// TIA Portal project "CIP" (V17)

(* hardware
DEVICE "S7-1200 station_1"  S7-1200 Station
   slot 0: "Rack_0"  S7-1200 Rack  Rack  V1.0
   slot 1: "PLC_1"  CPU 1214C DC/DC/DC  6ES7 214-1AG40-0XB0  V4.5
   slot 2: "AI 4x13BIT/AQ 2x14BIT_1"  6ES7 234-4HE32-0XB0  V2.1
   slot 3: "DI 16/DQ 16x24VDC_1"  6ES7 223-1BL32-0XB0  V2.0
DEVICE "HMI_1"  KTP600 Basic mono PN
   slot 0: "HMI_1"  KTP600 Basic mono PN  6AV6 647-0AB11-3AX0  12.0.0.0
   slot 1: "HMI_RT_1"  KTP600 Basic mono PN  6AV6 647-0AB11-3AX0  12.0.0.0
   slot 5: "HMI_1.IE_CP_1"  PROFINET Interface  12.0.0.0
      slot 1: "PROFINET Interface_1"  PROFINET Interface
         slot 1: "Port_1"  Port
*)

// ===== PLC "PLC_1"  CPU 1214C DC/DC/DC =====

VAR_GLOBAL   // PLC tag table "Default tag table"
   "VALVE_WASHABLE_DEVICE_INPUT" AT %Q1000.0 : Bool;
   "VALVE_WASHABLE_DEVICE_BACK" AT %Q1000.1 : Bool;
   "VALVE_INTERMEDIATE_1" AT %Q1000.2 : Bool;
   "VALVE_WATER_INPUT" AT %Q1000.3 : Bool;
   "VALVE_WATER_OUTPUT" AT %Q1000.4 : Bool;
   "VALVE_INTERMEDIATE_2" AT %Q1001.0 : Bool;
   "VALVE_INTERMEDIATE_3" AT %Q1001.1 : Bool;
   "VALVE_INTERMEDIATE_4" AT %Q1001.2 : Bool;
   "VALVE_WATER_TANK_INPUT" AT %Q1001.3 : Bool;
   "VALVE_WATER_TANK_INPUT_CLEAN" AT %Q1001.4 : Bool;
   "VALVE_WATER_TANK_OUTPUT" AT %Q1001.5 : Bool;
   "VALVE_ALKALI_TANK_INPUT" AT %Q1001.6 : Bool;
   "VALVE_ALKALI_TANK_INPUT_CLEAN" AT %Q1001.7 : Bool;
   "VALVE_ALKALI_TANK_OUTPUT" AT %Q1002.0 : Bool;
   "VALVE_ACID_TANK_INPUT" AT %Q1002.1 : Bool;
   "VALVE_ACID_TANK_INPUT_CLEAN" AT %Q1002.2 : Bool;
   "VALVE_ACID_TANK_OUTPUT" AT %Q1002.3 : Bool;
   "VALVE_STEAM" AT %Q1002.4 : Bool;
   "PUMP" AT %Q1002.5 : Bool;
   "BACK_PUMP" AT %Q1002.6 : Bool;
END_VAR

DATA_BLOCK "MAIN_DB"   // DB1
{ S7_Optimized_Access := 'TRUE' }
VERSION : 0.1
// stored: InstanceOfName MAIN
"MAIN"
BEGIN
END_DATA_BLOCK

DATA_BLOCK "ACTUATORS_DB"   // DB2
{ S7_Optimized_Access := 'TRUE' }
VERSION : 0.1
// stored: InstanceOfName ACTUATORS
"ACTUATORS"
BEGIN
END_DATA_BLOCK

DATA_BLOCK "VALVES_AND_PUMPS_STATES_DB"   // DB3
{ S7_Optimized_Access := 'TRUE' }
VERSION : 0.1
// stored: InstanceOfName VALVES_AND_PUMPS_STATES
"VALVES_AND_PUMPS_STATES"
BEGIN
END_DATA_BLOCK

FUNCTION_BLOCK "MAIN"   // FB1, SCL
{ S7_Optimized_Access := 'TRUE' }
VERSION : 0.1
BEGIN

   "VALVES_AND_PUMPS_STATES_DB"();

   "ACTUATORS_DB"();
END_FUNCTION_BLOCK

FUNCTION_BLOCK "ACTUATORS"   // FB2, SCL
{ S7_Optimized_Access := 'TRUE' }
VERSION : 0.1
   VAR
      VALVE_WASHABLE_DEVICE_INPUT : "ACTUATOR";
      VALVE_WASHABLE_DEVICE_BACK : "ACTUATOR";
      VALVE_INTERMEDIATE_1 : "ACTUATOR";
      VALVE_WATER_INPUT : "ACTUATOR";
      VALVE_WATER_OUTPUT : "ACTUATOR";
      VALVE_INTERMEDIATE_2 : "ACTUATOR";
      VALVE_INTERMEDIATE_3 : "ACTUATOR";
      VALVE_INTERMEDIATE_4 : "ACTUATOR";
      VALVE_WATER_TANK_INPUT : "ACTUATOR";
      VALVE_WATER_TANK_INPUT_CLEAN : "ACTUATOR";
      VALVE_WATER_TANK_OUTPUT : "ACTUATOR";
      VALVE_ALKALI_TANK_INPUT : "ACTUATOR";
      VALVE_ALKALI_TANK_INPUT_CLEAN : "ACTUATOR";
      VALVE_ALKALI_TANK_OUTPUT : "ACTUATOR";
      VALVE_ACID_TANK_INPUT : "ACTUATOR";
      VALVE_ACID_TANK_INPUT_CLEAN : "ACTUATOR";
      VALVE_ACID_TANK_OUTPUT : "ACTUATOR";
      VALVE_STEAM : "VALVE_STEAM1";
      PUMP : "ACTUATOR";
      BACK_PUMP : "ACTUATOR";
   END_VAR
BEGIN

   #VALVE_WASHABLE_DEVICE_INPUT("VALVE_WASHABLE_DEVICE_INPUT");

   #VALVE_WASHABLE_DEVICE_BACK("VALVE_WASHABLE_DEVICE_BACK");

   #VALVE_INTERMEDIATE_1("VALVE_INTERMEDIATE_1");

   #VALVE_WATER_INPUT("VALVE_WATER_INPUT");

   #VALVE_WATER_OUTPUT("VALVE_WATER_OUTPUT");

   #VALVE_INTERMEDIATE_2("VALVE_INTERMEDIATE_2");

   #VALVE_INTERMEDIATE_3("VALVE_INTERMEDIATE_3");

   #VALVE_INTERMEDIATE_4("VALVE_INTERMEDIATE_4");

   #VALVE_WATER_TANK_INPUT("VALVE_WATER_TANK_INPUT");

   #VALVE_WATER_TANK_INPUT_CLEAN("VALVE_WATER_TANK_INPUT_CLEAN");

   #VALVE_WATER_TANK_OUTPUT("VALVE_WATER_TANK_OUTPUT");

   #VALVE_ALKALI_TANK_INPUT("VALVE_ALKALI_TANK_INPUT");

   #VALVE_ALKALI_TANK_INPUT_CLEAN("VALVE_ALKALI_TANK_INPUT_CLEAN");

   #VALVE_ALKALI_TANK_OUTPUT("VALVE_ALKALI_TANK_OUTPUT");

   #VALVE_ACID_TANK_INPUT("VALVE_ACID_TANK_INPUT");

   #VALVE_ACID_TANK_INPUT_CLEAN("VALVE_ACID_TANK_INPUT_CLEAN");

   #VALVE_ACID_TANK_OUTPUT("VALVE_ACID_TANK_OUTPUT");

   #VALVE_STEAM();

   #PUMP("PUMP");

   #BACK_PUMP("BACK_PUMP");
END_FUNCTION_BLOCK

FUNCTION_BLOCK "ACTUATOR"   // FB3, SCL
{ S7_Optimized_Access := 'TRUE' }
VERSION : 0.1
   VAR_OUTPUT
      OUTPUT : Bool;
   END_VAR
   VAR
      MODE : Int;
      AUTO_VALUE : Bool;
   END_VAR
BEGIN
   CASE #MODE OF
       0:
           #OUTPUT := FALSE;
       1:
           #OUTPUT := TRUE;
       2:
           #OUTPUT := #AUTO_VALUE;
   END_CASE;
END_FUNCTION_BLOCK

FUNCTION_BLOCK "VALVES_AND_PUMPS_STATES"   // FB4, SCL
{ S7_Optimized_Access := 'TRUE' }
VERSION : 0.1
   VAR
      STATE : Int;
      VALVE_WASHABLE_DEVICE_BACK_STATES : Array[0..26] of Bool;
      VALVE_WASHABLE_DEVICE_INPUT_STATES : Array[0..26] of Bool;
      VALVE_INTERMEDIATE_1_STATES : Array[0..26] of Bool;
      VALVE_WATER_INPUT_STATES : Array[0..26] of Bool;
      VALVE_WATER_OUTPUT_STATES : Array[0..26] of Bool;
      VALVE_INTERMEDIATE_2_STATES : Array[0..26] of Bool;
      VALVE_INTERMEDIATE_3_STATES : Array[0..26] of Bool;
      VALVE_INTERMEDIATE_4_STATES : Array[0..26] of Bool;
      VALVE_WATER_TANK_INPUT_STATES : Array[0..26] of Bool;
      VALVE_WATER_TANK_INPUT_CLEAN_STATES : Array[0..26] of Bool;
      VALVE_WATER_TANK_OUTPUT_STATES : Array[0..26] of Bool;
      VALVE_ALKALI_TANK_INPUT_STATES : Array[0..26] of Bool;
      VALVE_ALKALI_TANK_INPUT_CLEAN_STATES : Array[0..26] of Bool;
      VALVE_ALKALI_TANK_OUTPUT_STATES : Array[0..26] of Bool;
      VALVE_ACID_TANK_INPUT_STATES : Array[0..26] of Bool;
      VALVE_ACID_TANK_INPUT_CLEAN_STATES : Array[0..26] of Bool;
      VALVE_ACID_TANK_OUTPUT_STATES : Array[0..26] of Bool;
      PUMP_STATES : Array[0..26] of Bool;
      BACK_PUMP_STATES : Array[0..26] of Bool;
   END_VAR
   // VALVE_WASHABLE_DEVICE_BACK_STATES[18] := TRUE;
   // VALVE_WASHABLE_DEVICE_BACK_STATES[19] := TRUE;
   // VALVE_WASHABLE_DEVICE_BACK_STATES[20] := TRUE;
   // VALVE_WASHABLE_DEVICE_BACK_STATES[24] := TRUE;
   // VALVE_WASHABLE_DEVICE_BACK_STATES[25] := TRUE;
   // VALVE_WASHABLE_DEVICE_BACK_STATES[26] := TRUE;
   // VALVE_WASHABLE_DEVICE_INPUT_STATES[15] := TRUE;
   // VALVE_WASHABLE_DEVICE_INPUT_STATES[16] := TRUE;
   // VALVE_WASHABLE_DEVICE_INPUT_STATES[17] := TRUE;
   // VALVE_WASHABLE_DEVICE_INPUT_STATES[21] := TRUE;
   // VALVE_WASHABLE_DEVICE_INPUT_STATES[22] := TRUE;
   // VALVE_WASHABLE_DEVICE_INPUT_STATES[23] := TRUE;
   // VALVE_INTERMEDIATE_1_STATES[1] := TRUE;
   // VALVE_INTERMEDIATE_1_STATES[2] := TRUE;
   // VALVE_INTERMEDIATE_1_STATES[3] := TRUE;
   // VALVE_INTERMEDIATE_1_STATES[4] := TRUE;
   // VALVE_INTERMEDIATE_1_STATES[5] := TRUE;
   // VALVE_INTERMEDIATE_1_STATES[6] := TRUE;
   // VALVE_INTERMEDIATE_1_STATES[7] := TRUE;
   // VALVE_INTERMEDIATE_1_STATES[8] := TRUE;
   // VALVE_INTERMEDIATE_1_STATES[9] := TRUE;
   // VALVE_INTERMEDIATE_1_STATES[10] := TRUE;
   // VALVE_INTERMEDIATE_1_STATES[11] := TRUE;
   // VALVE_INTERMEDIATE_1_STATES[12] := TRUE;
   // VALVE_INTERMEDIATE_1_STATES[13] := TRUE;
   // VALVE_INTERMEDIATE_1_STATES[14] := TRUE;
   // VALVE_INTERMEDIATE_1_STATES[15] := TRUE;
   // VALVE_INTERMEDIATE_1_STATES[16] := TRUE;
   // VALVE_INTERMEDIATE_1_STATES[17] := TRUE;
   // VALVE_INTERMEDIATE_1_STATES[18] := TRUE;
   // VALVE_INTERMEDIATE_1_STATES[19] := TRUE;
   // VALVE_INTERMEDIATE_1_STATES[20] := TRUE;
   // VALVE_INTERMEDIATE_1_STATES[21] := TRUE;
   // VALVE_INTERMEDIATE_1_STATES[22] := TRUE;
   // VALVE_INTERMEDIATE_1_STATES[23] := TRUE;
   // VALVE_INTERMEDIATE_1_STATES[24] := TRUE;
   // VALVE_INTERMEDIATE_1_STATES[25] := TRUE;
   // VALVE_INTERMEDIATE_1_STATES[26] := TRUE;
   // VALVE_WATER_INPUT_STATES[1] := TRUE;
   // VALVE_WATER_INPUT_STATES[2] := TRUE;
   // VALVE_WATER_INPUT_STATES[4] := TRUE;
   // VALVE_WATER_INPUT_STATES[5] := TRUE;
   // VALVE_WATER_INPUT_STATES[7] := TRUE;
   // VALVE_WATER_INPUT_STATES[8] := TRUE;
   // VALVE_WATER_INPUT_STATES[10] := TRUE;
   // VALVE_WATER_INPUT_STATES[11] := TRUE;
   // VALVE_WATER_INPUT_STATES[12] := TRUE;
   // VALVE_WATER_INPUT_STATES[13] := TRUE;
   // VALVE_WATER_INPUT_STATES[14] := TRUE;
   // VALVE_WATER_OUTPUT_STATES[12] := TRUE;
   // VALVE_WATER_OUTPUT_STATES[13] := TRUE;
   // VALVE_WATER_OUTPUT_STATES[14] := TRUE;
   // VALVE_INTERMEDIATE_2_STATES[1] := TRUE;
   // VALVE_INTERMEDIATE_2_STATES[2] := TRUE;
   // VALVE_INTERMEDIATE_2_STATES[3] := TRUE;
   // VALVE_INTERMEDIATE_2_STATES[4] := TRUE;
   // VALVE_INTERMEDIATE_2_STATES[5] := TRUE;
   // VALVE_INTERMEDIATE_2_STATES[6] := TRUE;
   // VALVE_INTERMEDIATE_2_STATES[7] := TRUE;
   // VALVE_INTERMEDIATE_2_STATES[8] := TRUE;
   // VALVE_INTERMEDIATE_2_STATES[9] := TRUE;
   // VALVE_INTERMEDIATE_2_STATES[10] := TRUE;
   // VALVE_INTERMEDIATE_2_STATES[11] := TRUE;
   // VALVE_INTERMEDIATE_2_STATES[12] := TRUE;
   // VALVE_INTERMEDIATE_2_STATES[13] := TRUE;
   // VALVE_INTERMEDIATE_2_STATES[14] := TRUE;
   // VALVE_INTERMEDIATE_2_STATES[15] := TRUE;
   // VALVE_INTERMEDIATE_2_STATES[16] := TRUE;
   // VALVE_INTERMEDIATE_2_STATES[17] := TRUE;
   // VALVE_INTERMEDIATE_2_STATES[18] := TRUE;
   // VALVE_INTERMEDIATE_2_STATES[19] := TRUE;
   // VALVE_INTERMEDIATE_2_STATES[20] := TRUE;
   // VALVE_INTERMEDIATE_2_STATES[21] := TRUE;
   // VALVE_INTERMEDIATE_2_STATES[22] := TRUE;
   // VALVE_INTERMEDIATE_2_STATES[23] := TRUE;
   // VALVE_INTERMEDIATE_2_STATES[24] := TRUE;
   // VALVE_INTERMEDIATE_2_STATES[25] := TRUE;
   // VALVE_INTERMEDIATE_2_STATES[26] := TRUE;
   // VALVE_INTERMEDIATE_3_STATES[1] := TRUE;
   // VALVE_INTERMEDIATE_3_STATES[2] := TRUE;
   // VALVE_INTERMEDIATE_3_STATES[3] := TRUE;
   // VALVE_INTERMEDIATE_3_STATES[4] := TRUE;
   // VALVE_INTERMEDIATE_3_STATES[5] := TRUE;
   // VALVE_INTERMEDIATE_3_STATES[6] := TRUE;
   // VALVE_INTERMEDIATE_3_STATES[7] := TRUE;
   // VALVE_INTERMEDIATE_3_STATES[8] := TRUE;
   // VALVE_INTERMEDIATE_3_STATES[9] := TRUE;
   // VALVE_INTERMEDIATE_3_STATES[10] := TRUE;
   // VALVE_INTERMEDIATE_3_STATES[11] := TRUE;
   // VALVE_INTERMEDIATE_3_STATES[12] := TRUE;
   // VALVE_INTERMEDIATE_3_STATES[13] := TRUE;
   // VALVE_INTERMEDIATE_3_STATES[14] := TRUE;
   // VALVE_INTERMEDIATE_3_STATES[15] := TRUE;
   // VALVE_INTERMEDIATE_3_STATES[16] := TRUE;
   // VALVE_INTERMEDIATE_3_STATES[17] := TRUE;
   // VALVE_INTERMEDIATE_3_STATES[18] := TRUE;
   // VALVE_INTERMEDIATE_3_STATES[19] := TRUE;
   // VALVE_INTERMEDIATE_3_STATES[20] := TRUE;
   // VALVE_INTERMEDIATE_3_STATES[21] := TRUE;
   // VALVE_INTERMEDIATE_3_STATES[22] := TRUE;
   // VALVE_INTERMEDIATE_3_STATES[23] := TRUE;
   // VALVE_INTERMEDIATE_3_STATES[24] := TRUE;
   // VALVE_INTERMEDIATE_3_STATES[25] := TRUE;
   // VALVE_INTERMEDIATE_3_STATES[26] := TRUE;
   // VALVE_INTERMEDIATE_4_STATES[1] := TRUE;
   // VALVE_INTERMEDIATE_4_STATES[2] := TRUE;
   // VALVE_INTERMEDIATE_4_STATES[3] := TRUE;
   // VALVE_INTERMEDIATE_4_STATES[4] := TRUE;
   // VALVE_INTERMEDIATE_4_STATES[5] := TRUE;
   // VALVE_INTERMEDIATE_4_STATES[6] := TRUE;
   // VALVE_INTERMEDIATE_4_STATES[7] := TRUE;
   // VALVE_INTERMEDIATE_4_STATES[8] := TRUE;
   // VALVE_INTERMEDIATE_4_STATES[9] := TRUE;
   // VALVE_INTERMEDIATE_4_STATES[10] := TRUE;
   // VALVE_INTERMEDIATE_4_STATES[11] := TRUE;
   // VALVE_INTERMEDIATE_4_STATES[12] := TRUE;
   // VALVE_INTERMEDIATE_4_STATES[13] := TRUE;
   // VALVE_INTERMEDIATE_4_STATES[14] := TRUE;
   // VALVE_INTERMEDIATE_4_STATES[15] := TRUE;
   // VALVE_INTERMEDIATE_4_STATES[16] := TRUE;
   // VALVE_INTERMEDIATE_4_STATES[17] := TRUE;
   // VALVE_INTERMEDIATE_4_STATES[18] := TRUE;
   // VALVE_INTERMEDIATE_4_STATES[19] := TRUE;
   // VALVE_INTERMEDIATE_4_STATES[20] := TRUE;
   // VALVE_INTERMEDIATE_4_STATES[21] := TRUE;
   // VALVE_INTERMEDIATE_4_STATES[22] := TRUE;
   // VALVE_INTERMEDIATE_4_STATES[23] := TRUE;
   // VALVE_INTERMEDIATE_4_STATES[24] := TRUE;
   // VALVE_INTERMEDIATE_4_STATES[25] := TRUE;
   // VALVE_INTERMEDIATE_4_STATES[26] := TRUE;
   // VALVE_WATER_TANK_INPUT_STATES[2] := TRUE;
   // VALVE_WATER_TANK_INPUT_STATES[3] := TRUE;
   // VALVE_WATER_TANK_INPUT_STATES[18] := TRUE;
   // VALVE_WATER_TANK_INPUT_STATES[24] := TRUE;
   // VALVE_WATER_TANK_INPUT_CLEAN_STATES[1] := TRUE;
   // VALVE_WATER_TANK_OUTPUT_STATES[3] := TRUE;
   // VALVE_WATER_TANK_OUTPUT_STATES[15] := TRUE;
   // VALVE_WATER_TANK_OUTPUT_STATES[21] := TRUE;
   // VALVE_ALKALI_TANK_INPUT_STATES[5] := TRUE;
   // VALVE_ALKALI_TANK_INPUT_STATES[6] := TRUE;
   // VALVE_ALKALI_TANK_INPUT_STATES[19] := TRUE;
   // VALVE_ALKALI_TANK_INPUT_STATES[25] := TRUE;
   // VALVE_ALKALI_TANK_INPUT_CLEAN_STATES[4] := TRUE;
   // VALVE_ALKALI_TANK_INPUT_CLEAN_STATES[12] := TRUE;
   // VALVE_ALKALI_TANK_INPUT_CLEAN_STATES[13] := TRUE;
   // VALVE_ALKALI_TANK_OUTPUT_STATES[6] := TRUE;
   // VALVE_ALKALI_TANK_OUTPUT_STATES[13] := TRUE;
   // VALVE_ALKALI_TANK_OUTPUT_STATES[16] := TRUE;
   // VALVE_ALKALI_TANK_OUTPUT_STATES[22] := TRUE;
   // VALVE_ACID_TANK_INPUT_STATES[8] := TRUE;
   // VALVE_ACID_TANK_INPUT_STATES[9] := TRUE;
   // VALVE_ACID_TANK_INPUT_STATES[11] := TRUE;
   // VALVE_ACID_TANK_INPUT_STATES[20] := TRUE;
   // VALVE_ACID_TANK_INPUT_STATES[26] := TRUE;
   // VALVE_ACID_TANK_INPUT_CLEAN_STATES[7] := TRUE;
   // VALVE_ACID_TANK_INPUT_CLEAN_STATES[14] := TRUE;
   // VALVE_ACID_TANK_OUTPUT_STATES[9] := TRUE;
   // VALVE_ACID_TANK_OUTPUT_STATES[14] := TRUE;
   // VALVE_ACID_TANK_OUTPUT_STATES[17] := TRUE;
   // VALVE_ACID_TANK_OUTPUT_STATES[23] := TRUE;
   // PUMP_STATES[1] := TRUE;
   // PUMP_STATES[2] := TRUE;
   // PUMP_STATES[3] := TRUE;
   // PUMP_STATES[4] := TRUE;
   // PUMP_STATES[5] := TRUE;
   // PUMP_STATES[6] := TRUE;
   // PUMP_STATES[7] := TRUE;
   // PUMP_STATES[8] := TRUE;
   // PUMP_STATES[9] := TRUE;
   // PUMP_STATES[10] := TRUE;
   // PUMP_STATES[11] := TRUE;
   // PUMP_STATES[12] := TRUE;
   // PUMP_STATES[13] := TRUE;
   // PUMP_STATES[14] := TRUE;
   // PUMP_STATES[15] := TRUE;
   // PUMP_STATES[16] := TRUE;
   // PUMP_STATES[17] := TRUE;
   // PUMP_STATES[18] := TRUE;
   // PUMP_STATES[19] := TRUE;
   // PUMP_STATES[20] := TRUE;
   // PUMP_STATES[21] := TRUE;
   // PUMP_STATES[22] := TRUE;
   // PUMP_STATES[23] := TRUE;
   // PUMP_STATES[24] := TRUE;
   // PUMP_STATES[25] := TRUE;
   // PUMP_STATES[26] := TRUE;
   // BACK_PUMP_STATES[24] := TRUE;
   // BACK_PUMP_STATES[25] := TRUE;
   // BACK_PUMP_STATES[26] := TRUE;
BEGIN
   "ACTUATORS_DB".VALVE_WASHABLE_DEVICE_BACK.AUTO_VALUE := #VALVE_WASHABLE_DEVICE_BACK_STATES[#STATE];
   "ACTUATORS_DB".VALVE_WASHABLE_DEVICE_INPUT.AUTO_VALUE := #VALVE_WASHABLE_DEVICE_INPUT_STATES[#STATE];
   "ACTUATORS_DB".VALVE_INTERMEDIATE_1.AUTO_VALUE := #VALVE_INTERMEDIATE_1_STATES[#STATE];
   "ACTUATORS_DB".VALVE_WATER_INPUT.AUTO_VALUE := #VALVE_WATER_INPUT_STATES[#STATE];
   "ACTUATORS_DB".VALVE_WATER_OUTPUT.AUTO_VALUE := #VALVE_WATER_OUTPUT_STATES[#STATE];
   "ACTUATORS_DB".VALVE_INTERMEDIATE_2.AUTO_VALUE := #VALVE_INTERMEDIATE_2_STATES[#STATE];
   "ACTUATORS_DB".VALVE_INTERMEDIATE_3.AUTO_VALUE := #VALVE_INTERMEDIATE_3_STATES[#STATE];
   "ACTUATORS_DB".VALVE_INTERMEDIATE_4.AUTO_VALUE := #VALVE_INTERMEDIATE_4_STATES[#STATE];
   "ACTUATORS_DB".VALVE_WATER_TANK_INPUT.AUTO_VALUE := #VALVE_WATER_TANK_INPUT_STATES[#STATE];
   "ACTUATORS_DB".VALVE_WATER_TANK_INPUT_CLEAN.AUTO_VALUE := #VALVE_WATER_TANK_INPUT_CLEAN_STATES[#STATE];
   "ACTUATORS_DB".VALVE_WATER_TANK_OUTPUT.AUTO_VALUE := #VALVE_WATER_TANK_OUTPUT_STATES[#STATE];
   "ACTUATORS_DB".VALVE_ALKALI_TANK_INPUT.AUTO_VALUE := #VALVE_ALKALI_TANK_INPUT_STATES[#STATE];
   "ACTUATORS_DB".VALVE_ALKALI_TANK_INPUT_CLEAN.AUTO_VALUE := #VALVE_ALKALI_TANK_INPUT_CLEAN_STATES[#STATE];
   "ACTUATORS_DB".VALVE_ALKALI_TANK_OUTPUT.AUTO_VALUE := #VALVE_ALKALI_TANK_OUTPUT_STATES[#STATE];
   "ACTUATORS_DB".VALVE_ACID_TANK_INPUT.AUTO_VALUE := #VALVE_ACID_TANK_INPUT_STATES[#STATE];
   "ACTUATORS_DB".VALVE_ACID_TANK_INPUT_CLEAN.AUTO_VALUE := #VALVE_ACID_TANK_INPUT_CLEAN_STATES[#STATE];
   "ACTUATORS_DB".VALVE_ACID_TANK_OUTPUT.AUTO_VALUE := #VALVE_ACID_TANK_OUTPUT_STATES[#STATE];
   "ACTUATORS_DB".PUMP.AUTO_VALUE := #PUMP_STATES[#STATE];
   "ACTUATORS_DB".BACK_PUMP.AUTO_VALUE := #BACK_PUMP_STATES[#STATE];
END_FUNCTION_BLOCK

FUNCTION_BLOCK "VALVE_STEAM1"   // FB5, SCL
{ S7_Optimized_Access := 'TRUE' }
VERSION : 0.1
   VAR
      MODE : Int;
      AUTO_VALUE : Bool;
   END_VAR
BEGIN

   //Добавить условие отключения при высокой температуре


   CASE #MODE OF
       0:
           "VALVE_STEAM" := FALSE;
       1:
           "VALVE_STEAM" := TRUE;
       2:
           "VALVE_STEAM" := #AUTO_VALUE;
   END_CASE;
END_FUNCTION_BLOCK

ORGANIZATION_BLOCK "MAIN_STUB"   // OB1, SCL, ProgramCycle
TITLE = "Main Program Sweep (Cycle)"
{ S7_Optimized_Access := 'TRUE' }
VERSION : 0.1
   VAR_INPUT
      Initial_Call : Bool;   // Initial call of this OB
      Remanence : Bool;   // =True, if remanent data are available
   END_VAR
BEGIN


   "MAIN_DB"();
END_ORGANIZATION_BLOCK

(* ===== HMI "HMI_RT_1" =====
system functions are stored by id; their names below are inferred from use
connection "HMI_Connection_1": ETHERNET, SMART_S7_1200_OMS

HMI tags "Default tag table"
   "Tag_ScreenNumber" : UInt, internal

Template "Template_1" 320x240
   Button "Exit" at 266,202 size 52x37; TextOff 'Exit'; PictureOff "ExitRuntime_KTP600_Basic_mono_PN"; PictureOn "ExitRuntime_KTP600_Basic_mono_PN"
      on Release: StopRuntime(0)
   Button "Template_Button" at 213,202 size 52x37; TextOff 'Text'
   Button "Template_Button_1" at 160,202 size 52x37; TextOff 'Text'
   Button "Template_Button_2" at 107,202 size 52x37; TextOff 'Text'
   Button "Alarms" at 54,202 size 52x37; TextOff 'Alarms'; PictureOff "AlarmDisplay_KTP600_Basic_mono_PN"; PictureOn "AlarmDisplay_KTP600_Basic_mono_PN"
      on Release: function_ef3f5d25("Alarm window_Unacknowledged", -1)
   Button "Start screen" at 1,202 size 52x37; TextOff 'Start screen'; PictureOff "NavigateHome_KTP600_Basic_mono_PN"; PictureOn "NavigateHome_KTP600_Basic_mono_PN"
      on Release: ActivateScreen("Root screen", 0)
   SymbolicIOField "Symbolic_IO_Field_Screen" at 69,7 size 164x24; TextOff '0'; TextOn '1'; TextList "TextList_ScreenNames"
      ProcessValue <- "Tag_ScreenNumber"
      on Change: ActivateScreenByNumber("Tag_ScreenNumber", 0)
   DateTimeField "HmiScreenItemData" at 235,19 size 85x19
   DateTimeField "HmiScreenItemData_1" at 235,0 size 85x19
   GraphicView "Logo" at 0,0 size 67x38; Picture "Logo of HMI_1"

screen "Root screen" 320x240, template "Template_1"
   on GenerateScreen: SetTag("Tag_ScreenNumber", 1)
   TextField "HmiScreenItemData" at 32,109 size 256x17; Text 'Welcome to HMI_1 (KTP600 Basic mono PN)!'
*)